FUNCTION_BLOCK FB_Barcoder IMPLEMENTS IStation
VAR_INPUT
END_VAR
VAR_OUTPUT
END_VAR
VAR
	bPartPresent				: BOOL;
	bReady						: BOOL;
	bBusy						: BOOL;
	
	StationState				: E_StationState;
	pPartStatus					: POINTER TO ST_PartStatus;
	
	rand						: DRAND;
	tmrWork						: TON;
	tmrDelay					: TON;
	sBarcode					: STRING(255);
END_VAR

PROPERTY Busy : BOOL
GET
END_GET
END_PROPERTY

METHOD Execute : PVOID
VAR
	
END_VAR
rand(Seed:=777);
CASE StationState OF
	
	E_StationState.IDLE:
		
		IF bPartPresent THEN
			tmrDelay(IN:=TRUE, PT:=T#250MS);
			IF tmrDelay.Q THEN
				tmrDelay(IN:=FALSE);
				StationState := E_StationState.WORKING;
			END_IF
		ELSE
			bReady := TRUE;
			bBusy := FALSE;
		END_IF
		
	E_StationState.WORKING:
		
		bReady := FALSE;
		bBusy := TRUE;
		
		tmrWork(IN:= TRUE, PT:=T#1.5S);
		IF tmrWork.Q THEN
			sBarcode := CONCAT('BRCD', TO_STRING(TO_DINT(rand.Num * 10000)));
			StationState := E_StationState.DONE;
			tmrWork(IN:=FALSE);
		END_IF
	
	E_StationState.DONE:
	
		bReady := TRUE;
		bBusy := FALSE;
		
		IF NOT bPartPresent THEN
			IF PartStatus <> 0 THEN
				PartStatus^.bBarcodeStatus := TRUE;
				PartStatus^.sBarcode := sBarcode;
			END_IF
			StationState := E_StationState.IDLE;
		END_IF
		
END_CASE
END_METHOD

PROPERTY Faulted : BOOL
GET
END_GET
END_PROPERTY

PROPERTY PartPresent : BOOL
GET
PartPresent := bPartPresent;
END_GET
END_PROPERTY

PROPERTY PartStatus : POINTER TO ST_PartStatus
GET
PartStatus := pPartStatus;
END_GET
SET
pPartStatus := PartStatus;
END_SET
END_PROPERTY

PROPERTY Ready : BOOL
GET
Ready := bReady;
END_GET
END_PROPERTY

END_FUNCTION_BLOCK

(* stored: Version 1.1.0.1, ProductVersion 3.1.4024.12
   POU FB_Barcoder: Id {aaabbb18-d528-4ab4-a05e-daf444c77711}, SpecialFunc None
   Property Busy: Id {c31e5f2e-ba36-4587-a1b2-6f357ddc97a5}
   Get Get: Id {4f31b199-67c9-4d06-ab37-6e4354bde33d}
   Method Execute: Id {1c1ca266-edb7-42e5-8d83-08cba2d9458b}
   Property Faulted: Id {0d0870f5-0a00-4a4a-887e-d2bbd0588e88}
   Get Get: Id {f612afdd-4ee9-49e1-a559-f9a6e67154cf}
   Property PartPresent: Id {7c81c14d-ea9c-4707-a919-45c8f2a74ef5}
   Get Get: Id {565257fb-af3d-4b8d-8e1b-81227c863d57}
   Property PartStatus: Id {d5b9566c-6b2c-4813-942e-3e13bde1d3ee}
   Get Get: Id {21baa63f-f129-437f-90f0-68fcfeb4b493}
   Set Set: Id {792e6a08-6ed8-4f6a-b09a-8010f73f2885}
   Property Ready: Id {024b54fb-0bcf-45f5-ac7f-6c8ba0ffd001}
   Get Get: Id {41c37775-2a9d-4440-871a-cb9cfb48740d} *)
